{attribute 'linkalways'} 
{attribute 'no_explicit_call' := 'This FB is a CLASS and must be accessed using methods or properties'}
{attribute 'enable_dynamic_creation'}
FUNCTION_BLOCK ABSTRACT Error IMPLEMENTS I_Error
VAR
END_VAR

PROPERTY ABSTRACT ErrorCode : UDINT
GET
END_GET
END_PROPERTY

PROPERTY PUBLIC ABSTRACT Message : T_MAXSTRING
GET
END_GET
END_PROPERTY

METHOD PROTECTED OnSerialize
VAR_INPUT
	Serializer : I_Serializer;
END_VAR
END_METHOD

METHOD PUBLIC SerializeWith
VAR_INPUT
	Serializer : I_Serializer;
END_VAR
Serializer.StartObject();
Serializer.AddKeyString('message',Message);
Serializer.AddKeyUdint('errorCode',ErrorCode);
OnSerialize(Serializer);
Serializer.EndObject();
END_METHOD

END_FUNCTION_BLOCK

(* stored: Version 1.1.0.1, ProductVersion 3.1.4024.12
   POU Error: Id {3515e40d-777d-086e-1dc5-e25dbbabd80a}, SpecialFunc None
   Folder Protected: Id {887f3b17-8e31-0b5c-2d86-65ac4f391b4a}
   Property ErrorCode: Id {443c9683-8c58-0776-1b0f-80ac57c3449b}
   Get Get: Id {02119e76-31be-01d2-02bf-96d7f11555ee}
   Property Message: Id {e2a32734-1d54-0a56-07cb-dfb54be1f349}
   Get Get: Id {dc55775d-b2bb-0231-3138-de763b7ce1cb}
   Method OnSerialize: Id {824b0a20-902e-0d1e-1725-0a5ec5992781}
   Method SerializeWith: Id {10c32aab-be5b-02bb-0000-71a31e6df822} *)
